(* CODESYS project Magazijn Structured Tekst 2V0 - Opdracht 2.project
   Company: Avans
   Description: Simulatie voor opstelling Sorteer Station.
   Title: Simulatie Sorteer Station
   Author: Rene Potters/Gerard Harkema
   Version: 0.1.0

Project tree, tasks and I/O mapping:
  Device : EHV-CPU1025, Hitachi-IES, order no. EHV-CPU1025, version 3.5.4.11
      settings: IP Address = '192.168.1.31'
    application MagazijnTestRealWorld
      libraries: Standard, * (System); Util, * (System); VisuDialogs, 3.5.12.0 (System)
      task MainTask (cyclic, interval t#20ms, priority 1) calls MagazijnTest
    Basic : Basic, Hitachi-IES, version 3.4.4.0
      <Empty>
      <Empty>
      <Empty>
      <Empty>
      <Empty>
      <Empty>
      <Empty>
      <Empty>
      <Empty>
      <Empty>
      <Empty>
  Device_1 : CODESYS Control Win V3, 3S - Smart Software Solutions GmbH, version 3.5.13.20
    application MagazijnTestSimulatie
      libraries: Standard, * (System); Util, * (System); VisuDialogs, 3.5.12.0 (System)
      task MainTask (cyclic, interval t#20ms, priority 1) calls MagazijnTest
      task Simulatie (cyclic, interval t#20ms, priority 1) calls MagazijnSim
  Simulatie/
    program MagazijnSim [ST]
    global variables SIM
    data type MagazijnDUT
  text list GlobalTextList
  Programma Structured Text/
    function block MagazijnClass [ST]
    TestProgramms/
      program MagazijnTest [ST]
    States/
      data type magazijnStates
  global variables GVL
  Visualisaties/
    visualisation BekerMagazijnHMI
*)

// Simulatie/MagazijnDUT
{attribute 'qualified_only'}
{attribute 'strict'}
TYPE MagazijnDUT :
(
	INGETROKKEN, INTREKKEN, UITGESTOTEN, UITSTOTEN, LEEG
);
END_TYPE

// Programma Structured Text/States/magazijnStates
// Datum : 17 december 2020, Auteur: Gerard Harkema
{attribute 'qualified_only'}
{attribute 'strict'}
TYPE magazijnStates :
(
	idle := 0,
	in,
	travel_out,
	out,
	travel_in,
	error
);
END_TYPE

// Simulatie/SIM
{attribute 'qualified_only'}
VAR_GLOBAL
	// Rotatie van de overzetter
	Vx_OvzRotate: INT := 0;
	// Visualisatie invisible blok
	Vx_OvzBlokLinks: BOOL := FALSE;
	// Visualisatie invisible blok
	Vx_OvzBlokOverzetter: BOOL := FALSE;
	// Visualisatie invisible blok
	Vx_OvzBlokRechts: BOOL := FALSE;
	// Visualisatie invisible blok
	Vx_OvzBlokGevallen: BOOL := FALSE;	
	// Magazijn opnieuw vullen (simulatie)
	Ix_MagazijnVullen 	: BOOL;
	// Goten legen (symulatie)
	Ix_GotenLegen	  	: BOOL;
	
	
	
	
	
	
	
	
	
	
	
	
	
	
	
	
	
	
	
	
	
	
	
	
	
	
	
	
	
	
	
	
	
	
	
	
	
	
	
	
	
	
	
	
	
	
	
	
	// Simulatie visualisatie 
	Vw_Rotate45: INT := 45;
	// Visualisatie X positie van de uitstoter
	Vw_MagUitstoterBekerX: INT := 30;
	// Visualisatie invisible blok uitgestoten
	Vx_MagBlokUit: BOOL := TRUE;
	// Visualisatie invisible blok 1
	Vx_MagBlok1: BOOL := TRUE;
	// Visualisatie invisible blok 2
	Vx_MagBlok2: BOOL := TRUE;
	// Visualisatie invisible blok 3
	Vx_MagBlok3: BOOL := TRUE;
	// Visualisatie invisible blok 4
	Vx_MagBlok4: BOOL := TRUE;
	// Visualisatie invisible blokken
	Vx_MagBlok: ARRAY[1..8] OF BOOL;
	// Aantal blokken in het magazijn
	Vw_MagBlokAantal: INT := 4;
	// Simulatie onthoudt dat een blok maar 1x wordt uitgestoten
	Vw_MagBlok1X: INT := 0;
	// Ligt er een blok op band
	Vw_SorBlokBand: BOOL := FALSE;
	// Rotatie van de stopper
	Vw_SorStopperRotate: INT := 0;
	// Rotatie van de stopper goot 1
	Vw_SorGoot1Rotate: INT := 0;
	// Rotatie van de stopper goot 2
	Vw_SorGoot2Rotate: INT := 0;
	// Kleur van de blok op betreffende positie
	Vw_SorKleurBand: DWORD := 0;
	// Bewegen van de blok over de band
	Vi_SorBlokBandX: INT := 0;
	// Bewegen van de blok over de band
	Vi_SorBlokBandY: INT := 0;
	// Simulatie error. Inverse logica.
	Vx_MagLuchtDrukError: BOOL := TRUE;
	// Simulatie error. Inverse logica.
	Vx_MagIsInError: BOOL := TRUE;
	// Simulatie error. Inverse logica.
	Vx_MagIsUitError: BOOL := TRUE;
	// Simulatie error. Inverse logica.
	Vx_OvzLuchtDrukError: BOOL := TRUE;
	// Simulatie error. Inverse logica.
	Vx_OvzIsLinksError: BOOL := TRUE;
	// Simulatie error. Inverse logica.
	Vx_OvzIsRechtsError: BOOL := TRUE;
	// Simulatie error. Inverse logica.
	Vx_OvzVacuumError: BOOL := TRUE;
	// Simulatie error. Inverse logica.
	Vx_SorMotorAfvoerError: BOOL := TRUE;
	// Simulatie error. Inverse logica.
	Vx_SorGoot1InError: BOOL := TRUE;
	// Simulatie error. Inverse logica.
	Vx_SorGoot1UitError: BOOL := TRUE;
	// Simulatie error. Inverse logica.
	Vx_SorInGootError: BOOL := TRUE;
	// Ligt er een blok op de betreffende positie
	Vx_SorBlokGoot: ARRAY [1..3,1..6] OF BOOL;
	// Kleur van de blok op betreffende positie
	Vw_SorKleurGoot: ARRAY [1..3,1..6] OF DWORD;
END_VAR

// GVL
VAR_GLOBAL
	// Indrukken resetknop 
	Ix_Resetknop: BOOL;
	// Keuzeknop staat op hand
	Ix_Hand: BOOL;
	// Keuzeknop staat op auto
	Ix_Auto: BOOL;
	// Indrukken noodstop
	Ix_Noodstop: BOOL;
	// Bekers magazijn zijn op
	Ix_MagazijnLeeg: BOOL;
	// Beker is uit dekselmagazijn gestoten
	Ix_UitstoterBekerIn: BOOL;
	// Uitstoter Beker haalt nieuwe beker op
	Ix_UitstoterBekerUit: BOOL;
	// Indrukken startknop
	Ix_Stopknop: BOOL := TRUE;
	// Indrukken stopknop
	Ix_Startknop: BOOL;	
	//Perslucht is aanwezig
	Ix_PersluchtAanwezig :BOOL;
	//Werkstuk door overzetter opgepakt
	Ix_VacuumAanwezig :BOOL;
	//Overzetter haalt beker op(linker pos.)
	Ix_OverzetterIsLinks :BOOL;
	//Overzetter plaatst beker op sorteerpositie
	Ix_OverzetterIsRechts :BOOL;
	//Beker aanwezig op detectiepositie
	Ix_BekerAanwezig :BOOL;
	//Beker is van aluminium
	Ix_BekerMetaal :BOOL;
	//Beker reflecteert en is dus niet zwart
	Ix_BekerReflecteerd :BOOL;
	//Product is naar een van de goten gegaan
	Ix_BekerInGoot :BOOL;
	//Pusher uitvoergoot 1 is in
	Ix_UitvoerGoot1IsIn :BOOL;
	//Pusher uitvoergoot 2 is in
	Ix_UitvoerGoot2IsIn :BOOL;
	//Beker afvoeren is bezig
	Ix_StationAfvoerVrij :BOOL;
	//Pusher uitvoergoot 1 is uit
	Ix_UitvoerGoot1IsUit :BOOL;
	//Pusher uitvoergoot 2 is uit
	Ix_UitvoerGoot2IsUit :BOOL;
	// Beker uit magazijn stoten
	Qx_BekerUitstoten: BOOL;	
	//Beker oppakken
	Qx_VacuumAan :BOOL;
	//Beker loslaten
	Qx_BekerLossen :BOOL;
	//Overzetter naar bekermagazijn
	Qx_OverzetterLinks :BOOL;
	//Overzetter naar sorteerpositie
	Qx_OverzetterRechts :BOOL;
	//Transportband aan
	Qx_MotorAfvoerAan :BOOL;
	//Pusher goot 1 uit
	Qx_UitvoerGoot1Uit :BOOL;
	//Pusher goot 2 uit
	Qx_UitvoerGoot2Uit :BOOL;
	//Beker stoppen op band voor detectie
	Qx_StopperUit :BOOL;
	//Uitsorteren is bezet
	Qx_StationBezet :BOOL;
	// Visualisatie invisible Gele vlak
	Qx_GeleLamp: BOOL;
	// Visualisatie invisible groene vlak
	Qx_GroeneLamp: BOOL;
	// Visualisatie invisible rode vlak
	Qx_RodeLamp: BOOL;
END_VAR

// Programma Structured Text/TestProgramms/MagazijnTest
// Datum : 17 december 2020, Auteur: Gerard Harkema
PROGRAM MagazijnTest
VAR
	xInitialaized				: BOOL := FALSE;
	
	// Bekers magazijn zijn op
	Ix_MagazijnLeegRef			: REFERENCE TO BOOL;
	// Beker is uit dekselmagazijn gestoten
	Ix_UitstoterBekerInRef		: REFERENCE TO BOOL;
	// Uitstoter Beker haalt nieuwe beker op
	Ix_UitstoterBekerUitRef		: REFERENCE TO BOOL;
	// Beker uit magazijn stoten
	Qx_BekerUitstotenRef		: REFERENCE TO BOOL;
	
	magazijn: MagazijnClass;
	
END_VAR

IF NOT xInitialaized THEN

	// Forse Persluct aanwezig
	gvl.Ix_PersluchtAanwezig := TRUE;
	
	xInitialaized	:= TRUE;
END_IF

IF Ix_Startknop THEN
	magazijn.start();
	Ix_Startknop := FALSE;
END_IF

IF Ix_Resetknop THEN
	magazijn.reset();
END_IF

IF Ix_Noodstop THEN
	magazijn.noodstop();
END_IF

Qx_GroeneLamp := magazijn.isKlaar();
Qx_RodeLamp := magazijn.isError();
Qx_GeleLamp := magazijn.isMagazijnLeeg();
 
magazijn.cycle();

END_PROGRAM

// Programma Structured Text/MagazijnClass
// Datum : 17 december 2020, Auteur: Gerard Harkema
FUNCTION_BLOCK MagazijnClass
VAR
	xInitialized				: BOOL := FALSE;
END_VAR

IF NOT xInitialized THEN

	xInitialized				:= TRUE;

END_IF

END_FUNCTION_BLOCK

// Simulatie/MagazijnSim
PROGRAM MagazijnSim
VAR
	// Timer om uitstoten en intrekken te vertragen
	Fb_Pulse: BLINK;
	// Timer om intrekken te vertragen
	Fb_Trigger: F_TRIG;
	// Eerste keer om visualisatie te updaten
	Mx_FirstTime: BOOL := TRUE;
	// Afhandeling van het magazijn
	Me_MagState: MAGAZIJNDUT := MAGAZIJNDUT.INGETROKKEN;
END_VAR

//
// Common stuff.
//

IF (Mx_FirstTime) THEN
	SIM.Vw_MagBlokAantal := 8;
	SIM.Vx_MagBlokUit:= FALSE;
	
	Mx_FirstTime := FALSE;
END_IF

					
//
// Handle all pulse and trigger events.
//
Fb_Pulse(ENABLE:=TRUE,TIMELOW:=T#200MS, TIMEHIGH:=T#200MS);
Fb_Trigger(CLK:=Fb_Pulse.OUT);


//
// Only if no emergency active, start handling the simulation.
//
IF (SIM.Ix_MagazijnVullen) THEN
	Mx_FirstTime := TRUE;
	SIM.Ix_MagazijnVullen := FALSE;
	RETURN;
END_IF
	
//
// The pulse determines the speed of the cilinder to move in
// ore move out. The cilinder is only moved if the airpressure 
// is available.
//
IF (Fb_Trigger.Q AND SIM.Vx_MagLuchtDrukError) THEN
		
			
	CASE Me_MagState OF
		MAGAZIJNDUT.INGETROKKEN:
			IF (SIM.Vx_MagBlokUit) THEN
				SIM.Vw_MagBlokAantal := SIM.Vw_MagBlokAantal - 1;
			END_IF
		
			SIM.Vw_MagUitstoterBekerX := 1;
			SIM.Vw_MagBlok1X    	  := SIM.Vw_MagUitstoterBekerX;
			SIM.Vx_MagBlokUit         := FALSE;
	
			IF (Qx_BekerUitstoten) THEN
				Me_MagState := MAGAZIJNDUT.UITSTOTEN;
			END_IF

		MAGAZIJNDUT.INTREKKEN:
			SIM.Vw_MagUitstoterBekerX := SIM.Vw_MagUitstoterBekerX - 30;
			
			IF (SIM.Vw_MagUitstoterBekerX < 0) THEN 
				SIM.Vw_MagUitstoterBekerX := 0; 
			END_IF		
			
			IF (SIM.Vw_MagUitstoterBekerX = 0) THEN
				Me_MagState := MAGAZIJNDUT.INGETROKKEN;				
			END_IF		

			IF (Qx_BekerUitstoten) THEN
				Me_MagState := MAGAZIJNDUT.UITSTOTEN;
			END_IF	
	
		MAGAZIJNDUT.UITGESTOTEN:
			SIM.Vx_MagBlokUit         := SIM.Vx_MagBlok1;
						
			IF (NOT Qx_BekerUitstoten) THEN
				Me_MagState := MAGAZIJNDUT.INTREKKEN;
			END_IF	
		
		MAGAZIJNDUT.UITSTOTEN:
			SIM.Vw_MagUitstoterBekerX := SIM.Vw_MagUitstoterBekerX + 30;
			SIM.Vw_MagBlok1X    	  := SIM.Vw_MagUitstoterBekerX;			
		
			IF (SIM.Vw_MagUitstoterBekerX > 70) THEN
				Me_MagState := MAGAZIJNDUT.UITGESTOTEN;				
			END_IF		

			IF (NOT Qx_BekerUitstoten) THEN
				Me_MagState := MAGAZIJNDUT.INTREKKEN;
			END_IF	
		
	END_CASE

	GVL.Ix_UitstoterBekerIn  := (Me_MagState = MAGAZIJNDUT.INGETROKKEN) AND SIM.Vx_MagIsInError;
	GVL.Ix_UitstoterBekerUit := (Me_MagState = MAGAZIJNDUT.UITGESTOTEN) AND SIM.Vx_MagIsUitError;	
	GVL.Ix_MagazijnLeeg 	 := (SIM.Vw_MagBlokAantal <= 0) AND (Ix_UitstoterBekerIn);	
	
	SIM.Vx_MagBlok[8] := (SIM.Vw_MagBlokAantal >= 8);
	SIM.Vx_MagBlok[7] := (SIM.Vw_MagBlokAantal >= 7);
	SIM.Vx_MagBlok[6] := (SIM.Vw_MagBlokAantal >= 6);
	SIM.Vx_MagBlok[5] := (SIM.Vw_MagBlokAantal >= 5);		
	SIM.Vx_MagBlok[4] := (SIM.Vw_MagBlokAantal >= 4);
	SIM.Vx_MagBlok[3] := (SIM.Vw_MagBlokAantal >= 3);
	SIM.Vx_MagBlok[2] := (SIM.Vw_MagBlokAantal >= 2);
	SIM.Vx_MagBlok[1] := (SIM.Vw_MagBlokAantal >= 1);	
	
END_IF

END_PROGRAM

// Visualisaties/BekerMagazijnHMI
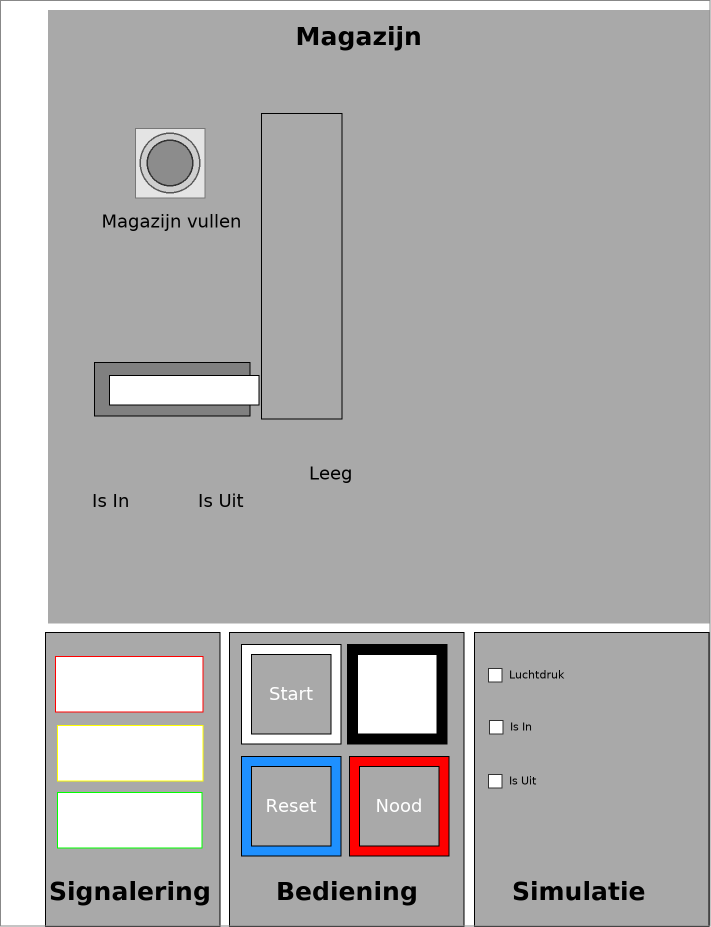
VISUALIZATION BekerMagazijnHMI  // 711x927
    Rectangle (47,9 664x615)
    Polygon (286,461) (316,461) (346,461) (376,461) (331,541), "Leeg", colour toggle: Ix_MagazijnLeeg
    Polygon (111,461) (111,461) (151,501) (111,541) (71,501), "Is In", colour toggle: Ix_UitstoterBekerIn
    Polygon (221,461) (221,461) (261,501) (221,541) (181,501), "Is Uit", colour toggle: Ix_UitstoterBekerUit
    Rectangle (94,362 156x54)
    Rectangle (261,113 81x306)
    Rectangle (353,376 61x29), colour toggle: SIM.Vx_MagBlokUit
    Rectangle (266,341 61x29), colour toggle: SIM.Vx_MagBlok[2]
    Rectangle (266,305 61x29), colour toggle: SIM.Vx_MagBlok[3]
    Rectangle (266,269 61x29), colour toggle: SIM.Vx_MagBlok[4]
    Rectangle (266,376 61x29), colour toggle: SIM.Vx_MagBlok[1]
        p3560616238: SIM.Vw_MagBlok1X
    Rectangle (109,375 150x30)
        p3560616238: SIM.Vw_MagUitstoterBekerX
    Label (284,21 150x30), "Magazijn"
    Group (45,632 664x295)
        Group (0,0 664x295)
            Group (429,0 235x295)
                Rectangle (0,0 235x295)
                Label (30,236 150x46), "Simulatie"
            Group (0,0 175x295)
                Rectangle (0,0 175x295)
                Rectangle (10,24 148x56), colour toggle: Qx_RodeLamp
                Rectangle (12,93 146x56), colour toggle: Qx_GeleLamp
                Rectangle (12,160 145x56), colour toggle: Qx_GroeneLamp
                Label (10,236 150x46), "Signalering"
            Group (184,0 235x295)
                Rectangle (0,0 235x295)
                Group (12,12 100x100)
                    RoundedRectangle (0,0 100x100)
                    RoundedRectangle (10,10 80x80), "Start", tooltip "Start knop", colour toggle: Ix_Startknop
                        OnMouseDown: execute { Ix_Startknop := TRUE; }
                        OnMouseUp: execute { Ix_Startknop := FALSE; }
                Group (118,12 100x100)
                    RoundedRectangle (0,0 100x100)
                    RoundedRectangle (10,10 80x80), "Stop", tooltip "Stop knop", colour toggle: Ix_Stopknop
                        OnMouseDown: execute { Ix_Stopknop := FALSE; }
                        OnMouseUp: execute { Ix_Stopknop := TRUE; }
                Group (12,124 100x100)
                    RoundedRectangle (0,0 100x100)
                    RoundedRectangle (10,10 80x80), "Reset", tooltip "Reset knop", colour toggle: Ix_Resetknop
                        OnMouseDown: execute { Ix_Resetknop := TRUE; }
                        OnMouseUp: execute { Ix_Resetknop := FALSE; }
                Group (120,124 100x100)
                    RoundedRectangle (0,0 100x100), "Nood"
                    RoundedRectangle (10,10 80x80), "Nood", tooltip "Noodstop", colour toggle: Ix_Noodstop
                        OnMouseDown: execute { Ix_Noodstop := NOT Ix_Noodstop; }
                Label (43,236 150x46), "Bediening"
        Checkbox (441,17 196x52), "Luchtdruk", variable: SIM.Vx_MagLuchtDrukError
        Checkbox (442,69 196x52), "Is In", variable: SIM.Vx_MagIsInError
        Checkbox (441,123 196x52), "Is Uit", variable: SIM.Vx_MagIsUitError
    Rectangle (266,197 61x29), colour toggle: SIM.Vx_MagBlok[6]
    Rectangle (266,161 61x29), colour toggle: SIM.Vx_MagBlok[7]
    Rectangle (266,125 61x29), colour toggle: SIM.Vx_MagBlok[8]
    Rectangle (266,232 61x29), colour toggle: SIM.Vx_MagBlok[5]
    PushSwitch (135,128 70x70), tooltip "Magazijn vullen", variable: SIM.Ix_MagazijnVullen, behaviour: TOGGLE, style: Switch-PushSwitch-Gray
    Polygon (94,209) (124,209) (154,209) (249,223) (149,237), "Magazijn vullen", colour toggle: Ix_MagazijnLeeg
END_VISUALIZATION
